Omron CX-Programmer project 新工程 (CX-Programmer 9.73)

# PLC 新PLC1: CP1H XA

## Global symbols (name address type ; comment)
1.00 BOOL  ; 南绿灯
1.01 BOOL  ; 南黄灯
1.02 BOOL  ; 南红灯
1.03 BOOL  ; 东西绿灯
1.04 BOOL  ; 东西黄灯
1.05 BOOL  ; 东西红灯

## Program 新程序1 (cyclic task 0)
; 该PLC的示例程序为城市十字路口设计的交通信号灯控制系统，适用于一个典型的四向交叉口。程序的核心是一个60秒的循环周期，确保交通灯的切换遵循固定的时间安排。南向和东西向各分配30秒的通行时间，绿灯亮起时允许车辆通行。在每个方向绿灯结束前的6秒，黄灯会闪烁，提醒驾驶员即将变灯。系统控制的物理设备包括南向的绿灯、黄灯、红灯，以及东西向的绿灯、黄灯、红灯。 / 实现逻辑： / 系统以秒计数器和每秒脉冲信号驱动时间每秒递增。 / 当秒计数器超过60秒时，自动重置为1，确保周期性。 / 下降沿检测标志检测每秒脉冲信号的下降沿。 / 系统运行标志配合下降沿检测标志驱动秒计数器每秒递增。 / 当秒计数器小于30秒时，南向绿灯控制和东西向红灯控制激活，允许南向车辆和行人通行，同时禁止东西向交通。 / 此时，东西向绿灯控制未激活。 / 当秒计数器进入24到30秒区间，且每秒脉冲信号为真时，南向黄灯控制开始每秒闪烁，同时南向绿灯控制熄灭，提醒驾驶员准备停车。 / 当秒计数器达到30秒或以上时，南向红灯控制亮起，禁止南向通行。 / 当秒计数器大于或等于30秒时，南向红灯控制和东西向绿灯控制激活，切换为东西向通行，同时南向绿灯控制和南向黄灯控制熄灭，南向交通停止。 / 接着，当秒计数器在54到60秒之间，且每秒脉冲信号为真时，东西向黄灯控制开始每秒闪烁，同时东西向绿灯控制熄灭，提示驾驶员准备停车。 / 整个过程中，南向黄灯控制和东西向黄灯控制不会同时闪烁，保证提示信号的唯一性。 / 当秒计数器小于30秒时，东西向红灯控制亮起，确保南向交通安全。
Local symbols
DO UINT

### Section 段1

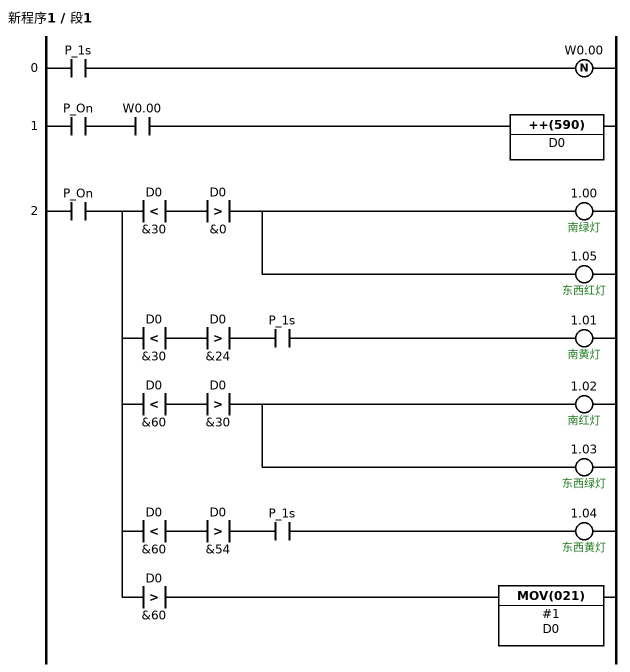
; rung 0
LD P_1s
DIFD(014) W0.00
; rung 1
LD P_On
AND W0.00
++(590) D0
; rung 2
LD P_On
OUT TR0
AND<(310) D0 &30
AND>(320) D0 &0
OUT 1.00  ; 南绿灯
OUT 1.05  ; 东西红灯
LD TR0
AND<(310) D0 &30
AND>(320) D0 &24
AND P_1s
OUT 1.01  ; 南黄灯
LD TR0
AND<(310) D0 &60
AND>(320) D0 &30
OUT 1.02  ; 南红灯
OUT 1.03  ; 东西绿灯
LD TR0
AND<(310) D0 &60
AND>(320) D0 &54
AND P_1s
OUT 1.04  ; 东西黄灯
LD TR0
AND>(320) D0 &60
MOV(021) #1 D0

### Section END
; rung 0
END(001)